RoboDK station: nozzle.rdk

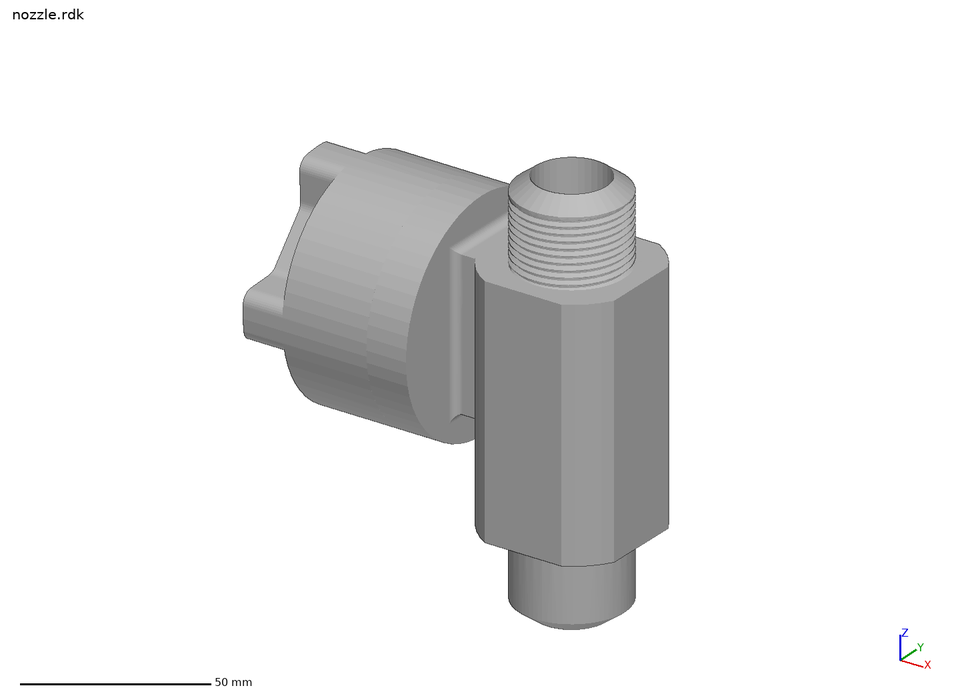
[picture v0: the station drawn from its stored meshes, robots at their saved joint values, targets as dots, program paths as lines]
Station nozzle (saved by RoboDK 5.5.4). Poses are relative to the parent item; angles as X-Y-Z fixed-axis rotations.
  - object end_effector_assembly_mod at (104, -5, -85) mm, rotated rx 90 ry 0 rz 0 deg, size 69.8 x 127 x 103.1 mm, geometry from end_effector_assembly_mod.STL
